TYPE TYP_RYG_TOWER_HW_OUT :
STRUCT
	Red AT %Q* : BOOL;
	Yellow AT %Q* : BOOL;
	Green AT %Q* : BOOL;
END_STRUCT
END_TYPE

(* stored: Version 1.1.0.1, ProductVersion 3.1.4024.12
   DUT TYP_RYG_TOWER_HW_OUT: Id {c3bd3904-3802-492d-8708-2bce8ec38818} *)
